PROGRAM Carga_semilla
VAR
	
	fbPE_H_VF1 :Equipo_Motor_ATV320;	//Elevador TRBB	
	fbPE_H_VF2 :Equipo_Motor_ATV320;	//Elevador carga tratadora
	Demora_PE_H_HLS: TON;
	Demora_TR_S_HLS: TON;
	ParadaPE_H_VF1: TOF;
	ParadaPE_TR_S_HLS: TOF;
	TmrDemoraPE_H_VF2: TOF;
	TmrDemoraPE_H_VF1: TOF;
	Tiempo_seg_to_TIME_PE_H_VF1: Tiempo_seg_to_TIME;
	Tiempo_seg_to_TIME_PE_H_VF2: Tiempo_seg_to_TIME;
	TDemoraTR_S_V7: TON;
	TDemoraTR_S_V8: TON;
END_VAR
VAR // added by the converter: edge detectors and wires of the graphical bodies
    _w1, _w2, _w3 : BOOL;
    _ft1, _ft2 : F_TRIG;
END_VAR

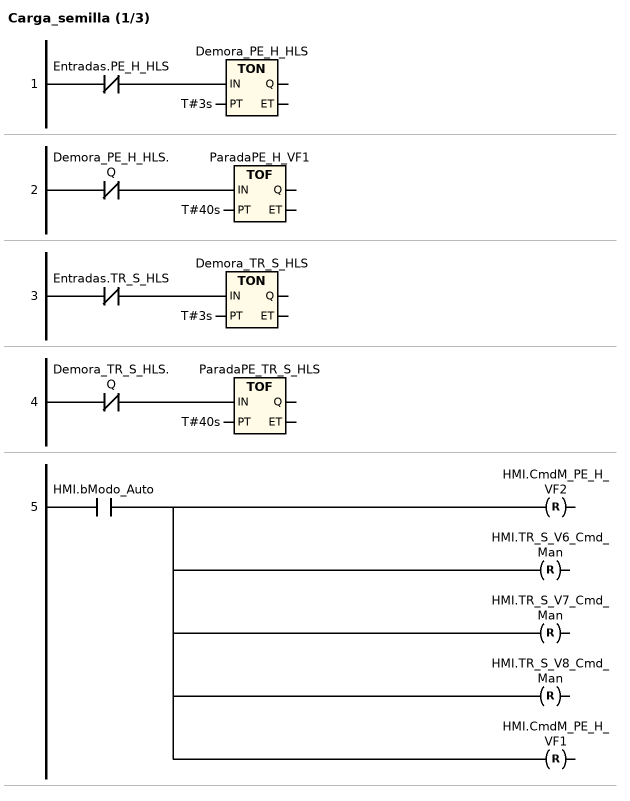
// NETWORK 1
Demora_PE_H_HLS(IN := NOT Entradas.PE_H_HLS, PT := T#3s); // TON

// NETWORK 2
ParadaPE_H_VF1(IN := NOT Demora_PE_H_HLS.Q, PT := T#40s); // TOF

// NETWORK 3
Demora_TR_S_HLS(IN := NOT Entradas.TR_S_HLS, PT := T#3s); // TON

// NETWORK 4
ParadaPE_TR_S_HLS(IN := NOT Demora_TR_S_HLS.Q, PT := T#40s); // TOF

// NETWORK 5
_w1 := HMI.bModo_Auto;
HMI.CmdM_PE_H_VF2 R= _w1;
HMI.TR_S_V6_Cmd_Man R= _w1;
HMI.TR_S_V7_Cmd_Man R= _w1;
HMI.TR_S_V8_Cmd_Man R= _w1;
HMI.CmdM_PE_H_VF1 R= _w1;

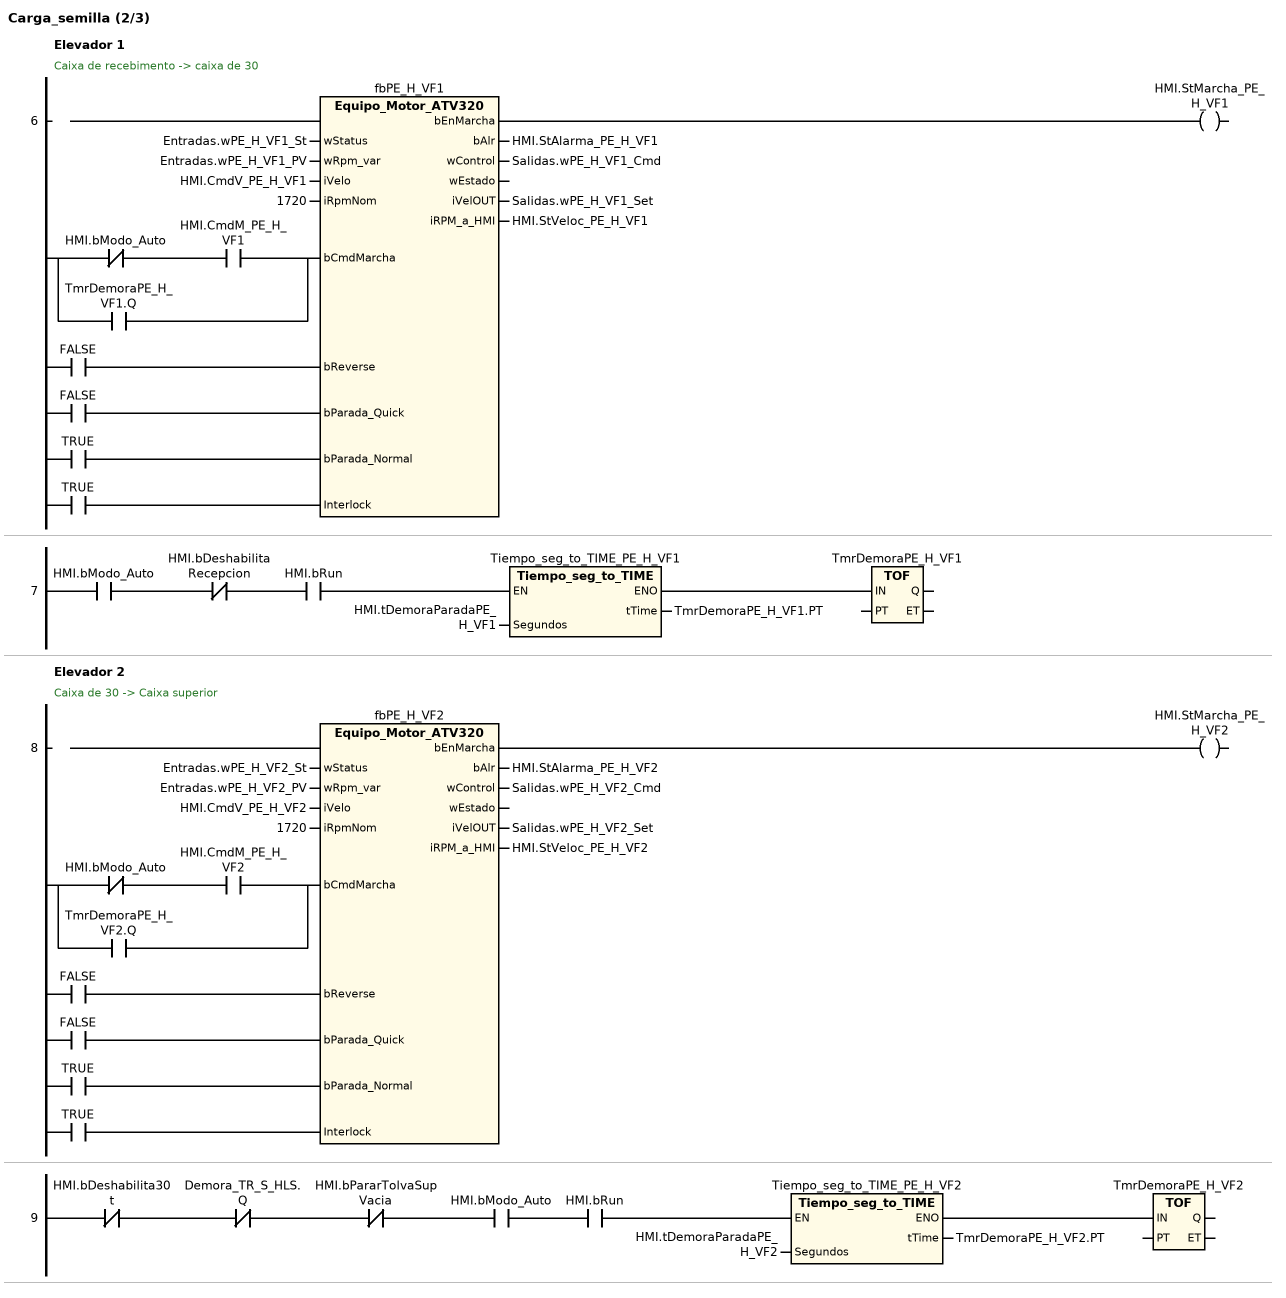
// NETWORK 6: Elevador 1
// Caixa de recebimento -> caixa de 30
fbPE_H_VF1(
    wStatus := Entradas.wPE_H_VF1_St,
    wRpm_var := Entradas.wPE_H_VF1_PV,
    iVelo := HMI.CmdV_PE_H_VF1,
    iRpmNom := 1720,
    bCmdMarcha := NOT HMI.bModo_Auto AND HMI.CmdM_PE_H_VF1 OR TmrDemoraPE_H_VF1.Q,
    bReverse := FALSE,
    bParada_Quick := FALSE,
    bParada_Normal := TRUE,
    Interlock := TRUE,
    bAlr => HMI.StAlarma_PE_H_VF1,
    wControl => Salidas.wPE_H_VF1_Cmd,
    iVelOUT => Salidas.wPE_H_VF1_Set,
    iRPM_a_HMI => HMI.StVeloc_PE_H_VF1); // Equipo_Motor_ATV320
HMI.StMarcha_PE_H_VF1 := fbPE_H_VF1.bEnMarcha;

// NETWORK 7
_w2 := HMI.bModo_Auto AND NOT HMI.bDeshabilitaRecepcion AND HMI.bRun;
IF _w2 THEN
    Tiempo_seg_to_TIME_PE_H_VF1(Segundos := HMI.tDemoraParadaPE_H_VF1, tTime => TmrDemoraPE_H_VF1.PT); // Tiempo_seg_to_TIME
END_IF
TmrDemoraPE_H_VF1(IN := _w2); // TOF

// NETWORK 8: Elevador 2
// Caixa de 30 -> Caixa superior
fbPE_H_VF2(
    wStatus := Entradas.wPE_H_VF2_St,
    wRpm_var := Entradas.wPE_H_VF2_PV,
    iVelo := HMI.CmdV_PE_H_VF2,
    iRpmNom := 1720,
    bCmdMarcha := NOT HMI.bModo_Auto AND HMI.CmdM_PE_H_VF2 OR TmrDemoraPE_H_VF2.Q,
    bReverse := FALSE,
    bParada_Quick := FALSE,
    bParada_Normal := TRUE,
    Interlock := TRUE,
    bAlr => HMI.StAlarma_PE_H_VF2,
    wControl => Salidas.wPE_H_VF2_Cmd,
    iVelOUT => Salidas.wPE_H_VF2_Set,
    iRPM_a_HMI => HMI.StVeloc_PE_H_VF2); // Equipo_Motor_ATV320
HMI.StMarcha_PE_H_VF2 := fbPE_H_VF2.bEnMarcha;

// NETWORK 9
_w3 := NOT HMI.bDeshabilita30t AND NOT Demora_TR_S_HLS.Q AND NOT HMI.bPararTolvaSupVacia AND HMI.bModo_Auto AND HMI.bRun;
IF _w3 THEN
    Tiempo_seg_to_TIME_PE_H_VF2(Segundos := HMI.tDemoraParadaPE_H_VF2, tTime => TmrDemoraPE_H_VF2.PT); // Tiempo_seg_to_TIME
END_IF
TmrDemoraPE_H_VF2(IN := _w3); // TOF

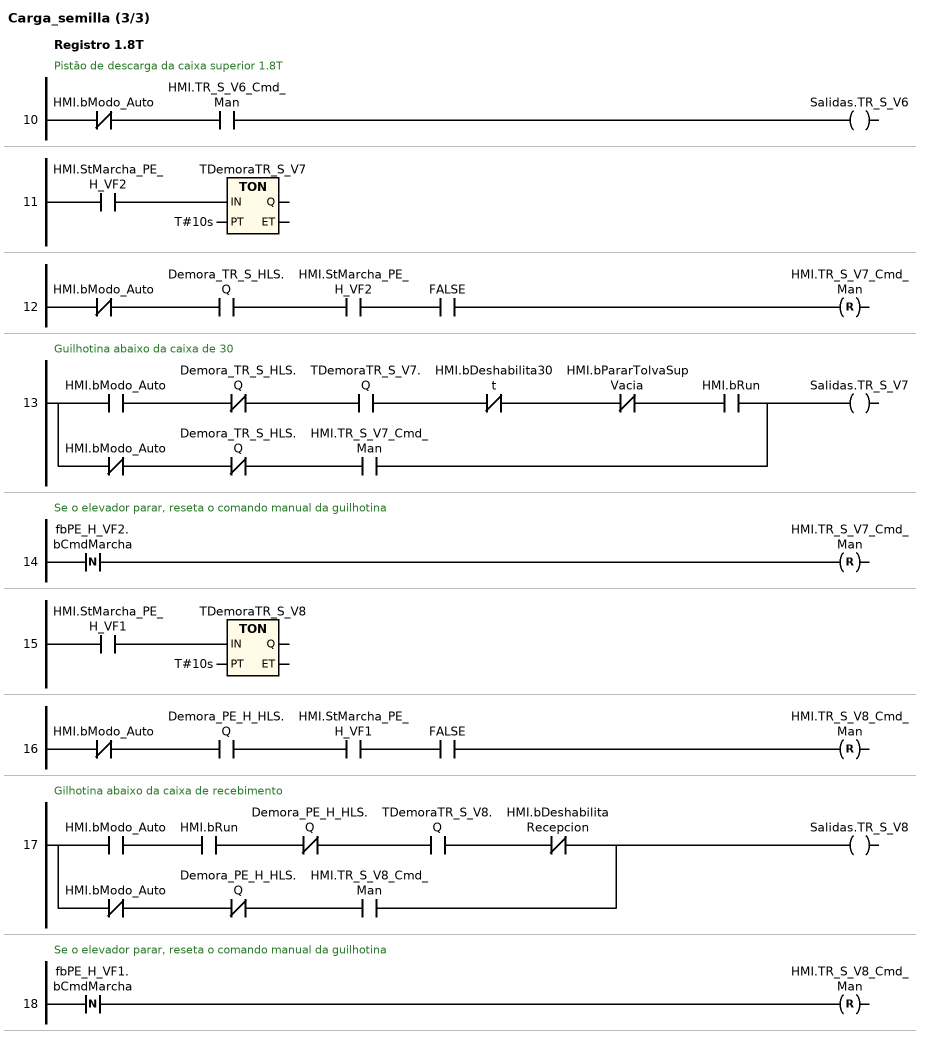
// NETWORK 10: Registro 1.8T
// Pistão de descarga da caixa superior 1.8T
Salidas.TR_S_V6 := NOT HMI.bModo_Auto AND HMI.TR_S_V6_Cmd_Man;

// NETWORK 11
TDemoraTR_S_V7(IN := HMI.StMarcha_PE_H_VF2, PT := T#10s); // TON

// NETWORK 12
HMI.TR_S_V7_Cmd_Man R= NOT HMI.bModo_Auto AND Demora_TR_S_HLS.Q AND HMI.StMarcha_PE_H_VF2 AND FALSE;

// NETWORK 13
// Guilhotina abaixo da caixa de 30
Salidas.TR_S_V7 := HMI.bModo_Auto AND NOT Demora_TR_S_HLS.Q AND TDemoraTR_S_V7.Q AND NOT HMI.bDeshabilita30t AND NOT HMI.bPararTolvaSupVacia AND HMI.bRun OR NOT HMI.bModo_Auto AND NOT Demora_TR_S_HLS.Q AND HMI.TR_S_V7_Cmd_Man;

// NETWORK 14
// Se o elevador parar, reseta o comando manual da guilhotina
_ft1(CLK := fbPE_H_VF2.bCmdMarcha);
HMI.TR_S_V7_Cmd_Man R= _ft1.Q;

// NETWORK 15
TDemoraTR_S_V8(IN := HMI.StMarcha_PE_H_VF1, PT := T#10s); // TON

// NETWORK 16
HMI.TR_S_V8_Cmd_Man R= NOT HMI.bModo_Auto AND Demora_PE_H_HLS.Q AND HMI.StMarcha_PE_H_VF1 AND FALSE;

// NETWORK 17
// Gilhotina abaixo da caixa de recebimento
Salidas.TR_S_V8 := HMI.bModo_Auto AND HMI.bRun AND NOT Demora_PE_H_HLS.Q AND TDemoraTR_S_V8.Q AND NOT HMI.bDeshabilitaRecepcion OR NOT HMI.bModo_Auto AND NOT Demora_PE_H_HLS.Q AND HMI.TR_S_V8_Cmd_Man;

// NETWORK 18
// Se o elevador parar, reseta o comando manual da guilhotina
_ft2(CLK := fbPE_H_VF1.bCmdMarcha);
HMI.TR_S_V8_Cmd_Man R= _ft2.Q;

END_PROGRAM

(* stored: Version 1.1.0.1, ProductVersion 3.1.4024.14
   POU Carga_semilla: Id {d40f2a46-10bc-457a-b5d9-1072047d8fb1}, SpecialFunc None *)
